FUNCTION_BLOCK EcMasterScanDevices IMPLEMENTS IEcTask
VAR_INPUT
END_VAR
VAR_OUTPUT
END_VAR
VAR
	iState : INT;
	masterScanDevices : Tc2_EtherCAT.FB_EcGetScannedSlaves;
	_scanDevices : ARRAY[0..Tc2_EtherCAT.EC_MAX_SLAVES] OF Tc2_EtherCAT.ST_EcSlaveScannedData;
	_execute: BOOL;
	_done: BOOL;
	_busy: BOOL;
	_error: BOOL;
	_netId: AMSNETID;
END_VAR

CASE iState OF
	0:
		IF _execute THEN
			_done := FALSE;
			_busy := TRUE;
			_error := FALSE;
			masterScanDevices.bExecute := TRUE;
			IF masterScanDevices.bBusy THEN
				iState := 10;
				_execute := false;
			END_IF
		END_IF
	10:
		IF NOT masterScanDevices.bBusy THEN
			IF NOT masterScanDevices.bError THEN
				_done := TRUE;
			ELSE
				_error := TRUE;
			END_IF
			_busy := FALSE;
			masterScanDevices.bExecute := FALSE;
			iState := 0;
		END_IF
END_CASE

masterScanDevices(sNetId := Tc2_System.F_CreateAmsNetId(nIds := NetId), 
					pArrEcScannedSlaveInfo := ADR(_scanDevices), 
					cbBufLen := SIZEOF(_scanDevices));

{warning 'add method implementation '}
METHOD Abort : BOOL
masterScanDevices.bExecute := FALSE;
_busy := FALSE;
_execute := FALSE;
Abort := TRUE;
iState := 0;
END_METHOD

{warning 'add property implementation'}
PROPERTY Busy : BOOL
GET
Busy := _busy;
END_GET
END_PROPERTY

{warning 'add property implementation'}
PROPERTY Done : BOOL
GET
Done := _done;
END_GET
END_PROPERTY

{warning 'add property implementation'}
PROPERTY Error : BOOL
GET
Error := _error;
END_GET
END_PROPERTY

{warning 'add method implementation '}
METHOD Execute : BOOL
IF NOT masterScanDevices.bBusy THEN
	Execute := _execute := true;
END_IF
END_METHOD

{warning 'add property implementation'}
PROPERTY NetID : amsnetid
GET
NetID := _netId;
END_GET
SET
_netId := NetID;
END_SET
END_PROPERTY

PROPERTY NumberScanDevices : udint
GET
NumberScanDevices := masterScanDevices.nSlaves;
END_GET
END_PROPERTY

PROPERTY ScannedDevices : reference to array[0..EC_MAX_Slaves] of ST_EcSlaveScannedData
GET
ScannedDevices REF= _scanDevices;
END_GET
END_PROPERTY

END_FUNCTION_BLOCK

(* stored: Version 1.1.0.1, ProductVersion 3.1.4024.11
   POU EcMasterScanDevices: Id {e9cf23b1-bc56-4e8a-9132-51e92ca67ec2}, SpecialFunc None
   Method Abort: Id {721f4d94-1f39-4958-980e-f9bad7204243}
   Property Busy: Id {e257315a-2c76-4a3a-862c-b8f1e65f2227}
   Get Get: Id {09f58fb5-4be0-41f3-bfb7-1fb866b25205}
   Property Done: Id {0176aa43-2e2d-48d0-9a44-330536bfcda1}
   Get Get: Id {c39d20d1-cc89-4ab7-b35b-668cd58f013c}
   Property Error: Id {6594d09c-f78e-41b5-bd66-f54b5b7c566b}
   Get Get: Id {f55cb9c0-f6a1-4bb5-bb4e-e7ab8a7e184b}
   Method Execute: Id {0af45555-7354-4edd-b7e6-387e2fb620e8}
   Property NetID: Id {cab19973-69d8-4521-b89a-48f6f2a85a27}
   Get Get: Id {40914e16-660e-4d88-b046-461ce326c266}
   Set Set: Id {a2660f98-a4dd-4435-b7da-cf6eb5e8f870}
   Property NumberScanDevices: Id {e2af7382-3e69-453d-882f-b90240b9f7ae}
   Get Get: Id {f2c25263-117f-4945-8c9e-7364c70d51d4}
   Property ScannedDevices: Id {72649964-0a1f-4333-a324-808f5f421d1a}
   Get Get: Id {efc35bb2-98cc-4980-8f38-29d8c7e9d00a} *)
